{attribute 'linkalways'} 
{attribute 'no_explicit_call' := 'This FB is a CLASS and must be accessed using methods or properties'}
{attribute 'enable_dynamic_creation'}
FUNCTION_BLOCK InstanceAddedEvent EXTENDS Event IMPLEMENTS I_InstanceAddedEvent
VAR
	_instance : I_Instance;
END_VAR

PROPERTY PUBLIC Instance : I_Instance
GET
Instance := _instance;
END_GET
END_PROPERTY

METHOD PUBLIC Notify
VAR_INPUT
	Instance : I_Instance;
END_VAR
_instance := Instance;
NotifySubscribers();
END_METHOD

END_FUNCTION_BLOCK

(* stored: Version 1.1.0.1, ProductVersion 3.1.4024.12
   POU InstanceAddedEvent: Id {35d6181b-52a3-070d-1198-f4b2cc71416e}, SpecialFunc None
   Property Instance: Id {107b830a-4f60-0f97-0343-5ed9afc76b3b}
   Get Get: Id {2c8a1ae2-6519-0f8a-00e8-0fc20ac22503}
   Method Notify: Id {b4bd003e-d157-093f-2255-c22be1aa6568} *)
